FUNCTION_BLOCK FB_Chamber1_Module EXTENDS FB_ModuleBase
VAR_INPUT	
	HwInput : ST_Chamber1_Signal_In;

	ServiceCtrl : REFERENCE TO ST_Chamber1_ServiceCtrl;
	ServiceParam : REFERENCE TO ST_Chamber1_ServiceParam;

	// Base unit used in Chamber1 chamber
	SpinAxis_BaseUnit : I_Axis_BaseUnit;
	LiftPinAxis_BaseUnit : I_Axis_BaseUnit;
END_VAR

VAR_OUTPUT
	HwOutput : ST_Chamber1_Signal_Out;
	ServiceStatus : ST_Chamber1_ServiceStatus;
END_VAR

VAR
	_EffectiveServiceCtrl : ST_Chamber1_ServiceCtrl;
	_EffectiveServiceParam : ST_Chamber1_ServiceParam;
	_ServiceStatusStore : ST_Chamber1_ServiceStatus;

	_SpinAxisJogCWService : FB_Chamber1SpinAxisJogCWServices;
	_SpinAxisMoveAbsService : FB_Chamber1SpinAxisMoveAbsServices;
	_SpinAxisMoveVelCWService : FB_Chamber1SpinAxisMoveVelCWServices;
	_LiftPinAxisMoveVelCWService : FB_Chamber1LiftPinAxisMoveVelCWServices;
	_LiftPinAxisMoveVelCCWService : FB_Chamber1LiftPinAxisMoveVelCCWServices;
	_LiftPinAxisMoveAbsService : FB_Chamber1LiftPinAxisMoveAbsServices;
	_SingleProcessService : FB_Chamber1SingleProcessService;
	_WaferSendService : FB_Chamber1WaferSendService;
	_WaferReceiveService : FB_Chamber1WaferReceiveService;

END_VAR

// An unbound Axis interface is a composition error. Keep the Module inert.
IF (SpinAxis_BaseUnit = 0) OR (LiftPinAxis_BaseUnit = 0) THEN
	RETURN;
END_IF

// Config wafer transfer endpoint
ModuleStatus.WaferTransferResponseList[1].EndpointId := 1;
ModuleStatus.WaferTransferResponseList[1].WaferHandlingType := E_WaferHandlingType.Passive;
ModuleStatus.WaferTransferResponseList[1].Capability := E_TransferCapability.Bidirectional;
ModuleStatus.WaferTransferResponseList[1].SendServiceId := E_Chamber1ServiceId.WaferSend;
ModuleStatus.WaferTransferResponseList[1].ReceiveServiceId := E_Chamber1ServiceId.WaferReceive;

M_UpdateModule();

// Update status
ServiceStatus := _ServiceStatusStore;

// Link status to module
ModuleStatus.WaferTransferResponseList[1].Send.Status := ServiceStatus.WaferSend;
ModuleStatus.WaferTransferResponseList[1].Send.Signal := _WaferSendService.SignalOut;
ModuleStatus.WaferTransferResponseList[1].SendReady := _ServiceCoordinator.AllIdle;
ModuleStatus.WaferTransferResponseList[1].Receive.Status := ServiceStatus.WaferReceive;
ModuleStatus.WaferTransferResponseList[1].Receive.Signal := _WaferReceiveService.SignalOut;
ModuleStatus.WaferTransferResponseList[1].ReceiveReady := _ServiceCoordinator.AllIdle;

METHOD PROTECTED H_RegisterServices
M_RegisterService(
	ServiceId := E_Chamber1ServiceId.SpinAxisJogCW,
	UpperCtrl := ServiceCtrl.SpinAxisJogCW,
	EffectiveCtrl := _EffectiveServiceCtrl.SpinAxisJogCW,
	UpperParam := ServiceParam.SpinAxisJogCW,
	EffectiveParam := _EffectiveServiceParam.SpinAxisJogCW,
	Status := _ServiceStatusStore.SpinAxisJogCW);
M_RegisterService(
	ServiceId := E_Chamber1ServiceId.SpinAxisMoveAbs,
	UpperCtrl := ServiceCtrl.SpinAxisMoveAbs,
	EffectiveCtrl := _EffectiveServiceCtrl.SpinAxisMoveAbs,
	UpperParam := ServiceParam.SpinAxisMoveAbs,
	EffectiveParam := _EffectiveServiceParam.SpinAxisMoveAbs,
	Status := _ServiceStatusStore.SpinAxisMoveAbs);
M_RegisterService(
	ServiceId := E_Chamber1ServiceId.SpinAxisMoveVelCW,
	UpperCtrl := ServiceCtrl.SpinAxisMoveVelCW,
	EffectiveCtrl := _EffectiveServiceCtrl.SpinAxisMoveVelCW,
	UpperParam := ServiceParam.SpinAxisMoveVelCW,
	EffectiveParam := _EffectiveServiceParam.SpinAxisMoveVelCW,
	Status := _ServiceStatusStore.SpinAxisMoveVelCW);
M_RegisterService(
	ServiceId := E_Chamber1ServiceId.LiftPinAxisMoveVelCW,
	UpperCtrl := ServiceCtrl.LiftPinAxisMoveVelCW,
	EffectiveCtrl := _EffectiveServiceCtrl.LiftPinAxisMoveVelCW,
	UpperParam := ServiceParam.LiftPinAxisMoveVelCW,
	EffectiveParam := _EffectiveServiceParam.LiftPinAxisMoveVelCW,
	Status := _ServiceStatusStore.LiftPinAxisMoveVelCW);
M_RegisterService(
	ServiceId := E_Chamber1ServiceId.LiftPinAxisMoveVelCCW,
	UpperCtrl := ServiceCtrl.LiftPinAxisMoveVelCCW,
	EffectiveCtrl := _EffectiveServiceCtrl.LiftPinAxisMoveVelCCW,
	UpperParam := ServiceParam.LiftPinAxisMoveVelCCW,
	EffectiveParam := _EffectiveServiceParam.LiftPinAxisMoveVelCCW,
	Status := _ServiceStatusStore.LiftPinAxisMoveVelCCW);
M_RegisterService(
	ServiceId := E_Chamber1ServiceId.LiftPinAxisMoveAbs,
	UpperCtrl := ServiceCtrl.LiftPinAxisMoveAbs,
	EffectiveCtrl := _EffectiveServiceCtrl.LiftPinAxisMoveAbs,
	UpperParam := ServiceParam.LiftPinAxisMoveAbs,
	EffectiveParam := _EffectiveServiceParam.LiftPinAxisMoveAbs,
	Status := _ServiceStatusStore.LiftPinAxisMoveAbs);
M_RegisterService(
	ServiceId := E_Chamber1ServiceId.WaferSend,
	UpperCtrl := ServiceCtrl.WaferSend,
	EffectiveCtrl := _EffectiveServiceCtrl.WaferSend,
	UpperParam := ServiceParam.WaferSend,
	EffectiveParam := _EffectiveServiceParam.WaferSend,
	Status := _ServiceStatusStore.WaferSend);
M_RegisterService(
	ServiceId := E_Chamber1ServiceId.WaferReceive,
	UpperCtrl := ServiceCtrl.WaferReceive,
	EffectiveCtrl := _EffectiveServiceCtrl.WaferReceive,
	UpperParam := ServiceParam.WaferReceive,
	EffectiveParam := _EffectiveServiceParam.WaferReceive,
	Status := _ServiceStatusStore.WaferReceive);
END_METHOD

METHOD PROTECTED H_UpdateBaseUnit
VAR_INPUT
END_VAR
SpinAxis_BaseUnit.M_CyclicUpdate();
LiftPinAxis_BaseUnit.M_CyclicUpdate();
END_METHOD

METHOD PROTECTED H_UpdateService
VAR_INPUT
END_VAR
_SpinAxisJogCWService(
	Ctrl:= _EffectiveServiceCtrl.SpinAxisJogCW,
	Param:= _EffectiveServiceParam.SpinAxisJogCW,
	Context:= _ServiceContext,
	Axis_BaseUnit:= SpinAxis_BaseUnit,
	// Owner IDs are assigned by the Module so each Service instance is unique.
	ServiceId:= E_Chamber1ServiceId.SpinAxisJogCW,
	Status=> _ServiceStatusStore.SpinAxisJogCW);

_SpinAxisMoveAbsService(
	Ctrl:= _EffectiveServiceCtrl.SpinAxisMoveAbs,
	Param:= _EffectiveServiceParam.SpinAxisMoveAbs,
	Context:= _ServiceContext,
	Axis_BaseUnit:= SpinAxis_BaseUnit,
	ServiceId:= E_Chamber1ServiceId.SpinAxisMoveAbs,
	Status=> _ServiceStatusStore.SpinAxisMoveAbs);

_SpinAxisMoveVelCWService(
	Ctrl:= _EffectiveServiceCtrl.SpinAxisMoveVelCW,
	Param:= _EffectiveServiceParam.SpinAxisMoveVelCW,
	Context:= _ServiceContext,
	Axis_BaseUnit:= SpinAxis_BaseUnit,
	ServiceId:= E_Chamber1ServiceId.SpinAxisMoveVelCW,
	Status=> _ServiceStatusStore.SpinAxisMoveVelCW);

_LiftPinAxisMoveVelCWService(
	Ctrl:= _EffectiveServiceCtrl.LiftPinAxisMoveVelCW,
	Param:= _EffectiveServiceParam.LiftPinAxisMoveVelCW,
	Context:= _ServiceContext,
	Axis_BaseUnit:= LiftPinAxis_BaseUnit,
	ServiceId:= E_Chamber1ServiceId.LiftPinAxisMoveVelCW,
	Status=> _ServiceStatusStore.LiftPinAxisMoveVelCW);

_LiftPinAxisMoveVelCCWService(
	Ctrl:= _EffectiveServiceCtrl.LiftPinAxisMoveVelCCW,
	Param:= _EffectiveServiceParam.LiftPinAxisMoveVelCCW,
	Context:= _ServiceContext,
	Axis_BaseUnit:= LiftPinAxis_BaseUnit,
	ServiceId:= E_Chamber1ServiceId.LiftPinAxisMoveVelCCW,
	Status=> _ServiceStatusStore.LiftPinAxisMoveVelCCW);

_LiftPinAxisMoveAbsService(
	Ctrl:= _EffectiveServiceCtrl.LiftPinAxisMoveAbs,
	Param:= _EffectiveServiceParam.LiftPinAxisMoveAbs,
	Context:= _ServiceContext,
	Axis_BaseUnit:= LiftPinAxis_BaseUnit,
	ServiceId:= E_Chamber1ServiceId.LiftPinAxisMoveAbs,
	Status=> _ServiceStatusStore.LiftPinAxisMoveAbs);

_SingleProcessService(
	Ctrl := ServiceCtrl.SingleProcess,
	Param:= ServiceParam.SingleProcess,
	Context := _ServiceContext,
	SpinAxis_BaseUnit := SpinAxis_BaseUnit,
	LiftPinAxis_BaseUnit := LiftPinAxis_BaseUnit,
	ServiceId := E_Chamber1ServiceId.SingleProcess,
	Status => _ServiceStatusStore.SingleProcess);

// Both directions share Station material and hardware storage.
// TODO: Coordinate Send/Receive access when implementing the transfer sequences.
_WaferSendService(
	Ctrl := _EffectiveServiceCtrl.WaferSend,
	Param := _EffectiveServiceParam.WaferSend,
	Context := _ServiceContext,
	ServiceId := E_Chamber1ServiceId.WaferSend,
	MaterialInfo := ModuleStatus.WaferTransferResponseList[1].MaterialInfo,
	SpinAxis_BaseUnit := SpinAxis_BaseUnit,
	LiftPinAxis_BaseUnit := LiftPinAxis_BaseUnit,
	Status => _ServiceStatusStore.WaferSend);

_WaferReceiveService(
	Ctrl := _EffectiveServiceCtrl.WaferReceive,
	Param := _EffectiveServiceParam.WaferReceive,
	Context := _ServiceContext,
	ServiceId := E_Chamber1ServiceId.WaferReceive,
	MaterialInfo := ModuleStatus.WaferTransferResponseList[1].MaterialInfo,
	SpinAxis_BaseUnit := SpinAxis_BaseUnit,
	LiftPinAxis_BaseUnit := LiftPinAxis_BaseUnit,
	Status => _ServiceStatusStore.WaferReceive);
END_METHOD

END_FUNCTION_BLOCK

(* stored: Version 1.1.0.1, ProductVersion 3.1.4026.18
   POU FB_Chamber1_Module: Id {d2b222b5-592d-46be-8a8e-fa50af509b93}, SpecialFunc None
   Folder ModuleUpdate: Id {a9f2fa3e-34f5-43fc-8823-0e0dbffba0ff}
   Method H_RegisterServices: Id {3d094774-a05b-4729-a18a-320af51f821a}
   Method H_UpdateBaseUnit: Id {23db425b-9082-4959-8f76-43820da7ead4}
   Method H_UpdateService: Id {fa65f410-1990-4021-8134-1329f3f00eeb} *)
